// TwinCAT 3 PLC project TcoTixonFeedingTests
// Title: TcoTixonFeedingTests
// Company: Vortex.Library
// Author: TcOpenGroup
// ProjectVersion: 0.6.0.913
// ProgramVersion: 3.1.4024.12
// libraries:
//   Tc2_Standard, * (Beckhoff Automation GmbH)
//   Tc2_System, * (Beckhoff Automation GmbH)
//   Tc3_Module, * (Beckhoff Automation GmbH)
//   TcoAbstractions, 0.6.0.913 (Vortex.Library)
//   TcoCore, 0.6.0.913 (Vortex.Library)
//   TcoIo, 0.6.0.913 (Vortex.Library)
//   TcoTixonFeeding, 0.6.0.913 (Vortex.Library)
//   TcoUtilities, 0.6.0.913 (Vortex.Library)
// project tree:
//   GVLs/ GVL.TcGVL, GVL_iXlinker.TcGVL
//   / PlcTask1.TcTTO
//   POUs/ MAIN.TcPOU
//   Tests/TcoContext/ eTypeOfTixon.TcDUT, SequenceTask.TcPOU, WpfContext.TcPOU
//   Tests/TcoTixonFeeding/ eTcoTixonFeedingSimpleTests.TcDUT, TcoTestContext.TcPOU, TcoTixonFeedingTest.TcPOU
//   DUTs/IO/PDOs/ Channel_830843C1.TcDUT, Channel_42CA91F7.TcDUT
//   DUTs/IO/Boxes/ EK1200_013D0B49.TcDUT, EL1008_78E8D3DD.TcDUT, EL2008_E2806B95.TcDUT, EL9011_D65D3D32.TcDUT
//   DUTs/IO/Devices/ SyncUnitTasks_5FDC9770.TcDUT, SyncUnits_C3A34B50.TcDUT
//   DUTs/IO/Topology/ EK1200_4A80C775.TcDUT, ECAT_x_A7FD7D81.TcDUT
// (motion and I/O tree: see PLC project tcotixonfeeding)
// real-time tasks:
//   TASK PlcTask: cycle T#10ms, priority 20, ADS port 350
//   TASK PlcTask1: cycle T#10ms, priority 1, ADS port 351
//   TASK PN: cycle T#8ms, priority 2, ADS port 301
// variable links:
//   TcoTixonFeedingTests/TcoTixonFeedingTests Instance <-> ECAT
//     PlcTask1 Inputs/GVL_iXlinker.ECAT_x.InfoData.AmsNetId <-> InfoData/AmsNetId
//     PlcTask1 Inputs/GVL_iXlinker.ECAT_x.InfoData.CfgSlaveCount <-> InfoData/CfgSlaveCount
//     PlcTask1 Inputs/GVL_iXlinker.ECAT_x.InfoData.ChangeCount <-> InfoData/ChangeCount
//     PlcTask1 Inputs/GVL_iXlinker.ECAT_x.InfoData.DevId <-> InfoData/DevId
//     PlcTask1 Inputs/GVL_iXlinker.ECAT_x.Inputs.DevState <-> Inputs/DevState
//     PlcTask1 Inputs/GVL_iXlinker.ECAT_x.Inputs.Frm0InputToggle <-> Inputs/Frm0InputToggle
//     PlcTask1 Inputs/GVL_iXlinker.ECAT_x.Inputs.Frm0State <-> Inputs/Frm0State
//     PlcTask1 Inputs/GVL_iXlinker.ECAT_x.Inputs.Frm0WcState <-> Inputs/Frm0WcState
//     PlcTask1 Inputs/GVL_iXlinker.ECAT_x.Inputs.SlaveCount <-> Inputs/SlaveCount
//     PlcTask1 Outputs/GVL_iXlinker.ECAT_x.Outputs.DevCtrl <-> Outputs/DevCtrl
//     PlcTask1 Outputs/GVL_iXlinker.ECAT_x.Outputs.Frm0Ctrl <-> Outputs/Frm0Ctrl
//     PlcTask1 Outputs/GVL_iXlinker.ECAT_x.Outputs.Frm0WcCtrl <-> Outputs/Frm0WcCtrl
//   TcoTixonFeedingTests/TcoTixonFeedingTests Instance <-> ECAT/EK1200/IA1
//     PlcTask1 Inputs/GVL_iXlinker.ECAT_x.EK1200.IA1.Channel_{1..8}.Input <-> Channel {1..8}/Input  (8 links)
//     PlcTask1 Inputs/GVL_iXlinker.ECAT_x.EK1200.IA1.InfoData.State <-> InfoData/State
//     PlcTask1 Inputs/GVL_iXlinker.ECAT_x.EK1200.IA1.WcState.InputToggle <-> WcState/InputToggle
//     PlcTask1 Inputs/GVL_iXlinker.ECAT_x.EK1200.IA1.WcState.WcState <-> WcState/WcState
//   TcoTixonFeedingTests/TcoTixonFeedingTests Instance <-> ECAT/EK1200/QA1
//     PlcTask1 Inputs/GVL_iXlinker.ECAT_x.EK1200.QA1.InfoData.State <-> InfoData/State
//     PlcTask1 Inputs/GVL_iXlinker.ECAT_x.EK1200.QA1.WcState.WcState <-> WcState/WcState
//     PlcTask1 Outputs/GVL_iXlinker.ECAT_x.EK1200.QA1.Channel_{1..8}.Output <-> Channel {1..8}/Output  (8 links)

CONFIGURATION TcoTixonFeedingTests
    RESOURCE PLC ON TwinCAT3
        TASK PlcTask1(INTERVAL := T#10ms, PRIORITY := 1);
        PROGRAM MAIN WITH PlcTask1 : MAIN;
    END_RESOURCE
END_CONFIGURATION

// ---- Tests/TcoContext/eTypeOfTixon.TcDUT
{attribute 'qualified_only'}
{attribute 'strict'}
TYPE eTypeOfTixon :
(
    TixonStep := 0,
    TixonVibro := 1,
    TixonPickStep := 2,
    TixonPickVibro := 3,
    TixonPickVibroBasic := 4
);
END_TYPE

// ---- Tests/TcoTixonFeeding/eTcoTixonFeedingSimpleTests.TcDUT
{attribute 'qualified_only'}
{attribute 'strict'}
TYPE eTcoTixonFeedingSimpleTests :
(
    Restore := 1,
    CleanUp,
    Message,
    PowerDisable,
    PowerEnable,
    Reset,
    Last
);
END_TYPE

// ---- DUTs/IO/PDOs/Channel_830843C1.TcDUT
{attribute 'GeneratedUsingTerminal: EL1008-0000-0018'}
{attribute addProperty BoxType "EL1008-0000-0018"}
{attribute addProperty Id "InputAT %I*BOOL1"}
{attribute addProperty CRC "2198356929"}
{attribute addProperty Size "1"}
TYPE Channel_830843C1 EXTENDS TcoIo.InputBase_8311D824 :
STRUCT
    {attribute addProperty Name "Input"}
    Input AT %I* : BOOL;
END_STRUCT
END_TYPE

// ---- DUTs/IO/PDOs/Channel_42CA91F7.TcDUT
{attribute 'GeneratedUsingTerminal: EL2008-0000-0018'}
{attribute addProperty BoxType "EL2008-0000-0018"}
{attribute addProperty Id "OutputAT %Q*BOOL1"}
{attribute addProperty CRC "1120571895"}
{attribute addProperty Size "1"}
TYPE Channel_42CA91F7 EXTENDS TcoIo.OutputBase_10CEE7DE :
STRUCT
    {attribute addProperty Name "Output"}
    Output AT %Q* : BOOL;
END_STRUCT
END_TYPE

// ---- DUTs/IO/Boxes/EK1200_013D0B49.TcDUT
{attribute 'GeneratedUsingTerminal: EK1200-1388-0000'}
{attribute addProperty VendorId "#x00000002"}
{attribute addProperty BoxType "EK1200-1388-0000"}
{attribute addProperty Description "EK1200-5000 EtherCAT Power supply (2A E-Bus)"}
{attribute addProperty Physics "YK"}
{attribute addProperty Id "EK1200"}
{attribute addProperty CRC "20777801"}
{attribute addProperty Size "0"}
TYPE EK1200_013D0B49 EXTENDS TcoIo.EtcSlaveBoxBase_77A0E4A7 :
STRUCT
END_STRUCT
END_TYPE

// ---- DUTs/IO/Boxes/EL1008_78E8D3DD.TcDUT
{attribute 'GeneratedUsingTerminal: EL1008-0000-0018'}
{attribute addProperty VendorId "#x00000002"}
{attribute addProperty BoxType "EL1008-0000-0018"}
{attribute addProperty Description "EL1008 8Ch. Dig. Input 24V, 3ms"}
{attribute addProperty Physics "KK"}
{attribute addProperty Id "Channel_1AT %I*Channel_830843C11Channel_2AT %I*Channel_830843C11Channel_3AT %I*Channel_830843C11Channel_4AT %I*Channel_830843C11Channel_5AT %I*Channel_830843C11Channel_6AT %I*Channel_830843C11Channel_7AT %I*Channel_830843C11Channel_8AT %I*Channel_830843C11WcStateAT %I*WcState_9091E0EB2InfoDataAT %I*InfoData_6F19DB2B2"}
{attribute addProperty CRC "2028524509"}
{attribute addProperty Size "12"}
TYPE EL1008_78E8D3DD EXTENDS TcoIo.EtcSlaveTerminalBase_947E5A46 :
STRUCT
    {attribute addProperty Name "Channel_1"}
    Channel_1 : Channel_830843C1;
    {attribute addProperty Name "Channel_2"}
    Channel_2 : Channel_830843C1;
    {attribute addProperty Name "Channel_3"}
    Channel_3 : Channel_830843C1;
    {attribute addProperty Name "Channel_4"}
    Channel_4 : Channel_830843C1;
    {attribute addProperty Name "Channel_5"}
    Channel_5 : Channel_830843C1;
    {attribute addProperty Name "Channel_6"}
    Channel_6 : Channel_830843C1;
    {attribute addProperty Name "Channel_7"}
    Channel_7 : Channel_830843C1;
    {attribute addProperty Name "Channel_8"}
    Channel_8 : Channel_830843C1;
    {attribute addProperty Name "WcState"}
    WcState : TcoIo.WcState_9091E0EB;
    {attribute addProperty Name "InfoData"}
    InfoData : TcoIo.InfoData_6F19DB2B;
END_STRUCT
END_TYPE

// ---- DUTs/IO/Boxes/EL2008_E2806B95.TcDUT
{attribute 'GeneratedUsingTerminal: EL2008-0000-0018'}
{attribute addProperty VendorId "#x00000002"}
{attribute addProperty BoxType "EL2008-0000-0018"}
{attribute addProperty Description "EL2008 8Ch. Dig. Output 24V, 0.5A"}
{attribute addProperty Physics "KK"}
{attribute addProperty Id "Channel_1AT %Q*Channel_42CA91F71Channel_2AT %Q*Channel_42CA91F71Channel_3AT %Q*Channel_42CA91F71Channel_4AT %Q*Channel_42CA91F71Channel_5AT %Q*Channel_42CA91F71Channel_6AT %Q*Channel_42CA91F71Channel_7AT %Q*Channel_42CA91F71Channel_8AT %Q*Channel_42CA91F71WcStateAT %I*WcState_0B2B16F91InfoDataAT %I*InfoData_6F19DB2B2"}
{attribute addProperty CRC "3800066965"}
{attribute addProperty Size "11"}
TYPE EL2008_E2806B95 EXTENDS TcoIo.EtcSlaveTerminalBase_947E5A46 :
STRUCT
    {attribute addProperty Name "Channel_1"}
    Channel_1 : Channel_42CA91F7;
    {attribute addProperty Name "Channel_2"}
    Channel_2 : Channel_42CA91F7;
    {attribute addProperty Name "Channel_3"}
    Channel_3 : Channel_42CA91F7;
    {attribute addProperty Name "Channel_4"}
    Channel_4 : Channel_42CA91F7;
    {attribute addProperty Name "Channel_5"}
    Channel_5 : Channel_42CA91F7;
    {attribute addProperty Name "Channel_6"}
    Channel_6 : Channel_42CA91F7;
    {attribute addProperty Name "Channel_7"}
    Channel_7 : Channel_42CA91F7;
    {attribute addProperty Name "Channel_8"}
    Channel_8 : Channel_42CA91F7;
    {attribute addProperty Name "WcState"}
    WcState : TcoIo.WcState_0B2B16F9;
    {attribute addProperty Name "InfoData"}
    InfoData : TcoIo.InfoData_6F19DB2B;
END_STRUCT
END_TYPE

// ---- DUTs/IO/Boxes/EL9011_D65D3D32.TcDUT
{attribute 'GeneratedUsingTerminal: EL9011--0000'}
{attribute addProperty VendorId "#x00000002"}
{attribute addProperty BoxType "EL9011--0000"}
{attribute addProperty Description "EL9011 End Terminal"}
{attribute addProperty Physics ""}
{attribute addProperty Id "EL9011"}
{attribute addProperty CRC "3596434738"}
{attribute addProperty Size "0"}
TYPE EL9011_D65D3D32 EXTENDS TcoIo.EtcSlaveEndTerminalBase_866C7F0C :
STRUCT
END_STRUCT
END_TYPE

// ---- DUTs/IO/Devices/SyncUnitTasks_5FDC9770.TcDUT
{attribute 'GeneratedUsingTerminal: '}
{attribute addProperty BoxType ""}
{attribute addProperty Id "unreferencedAT %I*SyncUnitTask_AB2F50799PlcTask1AT %I*SyncUnitTask_AB2F50799"}
{attribute addProperty CRC "1608292208"}
{attribute addProperty Size "18"}
TYPE SyncUnitTasks_5FDC9770 EXTENDS TcoIo.SyncUnitTasksBase_7C8711EB :
STRUCT
    {attribute addProperty Name "unreferenced"}
    unreferenced : TcoIo.SyncUnitTask_AB2F5079;
    {attribute addProperty Name "PlcTask1"}
    PlcTask1 : TcoIo.SyncUnitTask_AB2F5079;
END_STRUCT
END_TYPE

// ---- DUTs/IO/Devices/SyncUnits_C3A34B50.TcDUT
{attribute 'GeneratedUsingTerminal: '}
{attribute addProperty BoxType ""}
{attribute addProperty Id "_defaultAT %I*SyncUnitTasks_5FDC977018"}
{attribute addProperty CRC "3282258768"}
{attribute addProperty Size "18"}
TYPE SyncUnits_C3A34B50 EXTENDS TcoIo.SyncUnitsBase_AD6C35CE :
STRUCT
    {attribute addProperty Name "_default"}
    _default : SyncUnitTasks_5FDC9770;
END_STRUCT
END_TYPE

// ---- DUTs/IO/Topology/EK1200_4A80C775.TcDUT
{attribute 'GeneratedUsingTerminal: EK1200-1388-0000'}
{attribute addProperty BoxType "EK1200-1388-0000"}
{attribute addProperty Id "IA1EL1008_78E8D3DD12QA1EL2008_E2806B9511Term_4_EL9011EL9011_D65D3D320"}
{attribute addProperty CRC "1249953653"}
{attribute addProperty Size "23"}
{attribute addProperty Name "EK1200"}
TYPE EK1200_4A80C775 EXTENDS EK1200_013D0B49 :
STRUCT
    {attribute addProperty Name "IA1"}
    {attribute addProperty PreviousPort "EK1200 : B"}
    {attribute addProperty SyncUnit "default"}
    IA1 : EL1008_78E8D3DD;
    {attribute addProperty Name "QA1"}
    {attribute addProperty PreviousPort "IA1 : B"}
    {attribute addProperty SyncUnit "default"}
    QA1 : EL2008_E2806B95;
    {attribute addProperty Name "Term 4 (EL9011)"}
    {attribute addProperty PreviousPort "QA1 : B"}
    {attribute addProperty SyncUnit "default"}
    Term_4_EL9011 : EL9011_D65D3D32;
END_STRUCT
END_TYPE

// ---- DUTs/IO/Topology/ECAT_x_A7FD7D81.TcDUT
{attribute 'GeneratedUsingTerminal: IODEVICETYPE_ETHERCATPROT'}
{attribute addProperty BoxType "IODEVICETYPE_ETHERCATPROT"}
{attribute addProperty Id "EK1200EK1200_4A80C77523SyncUnitsSyncUnits_C3A34B5018InputsInputs_A65FACA410OutputsOutputs_23C0ED1D6InfoDataInfoData_84133AC922"}
{attribute addProperty CRC "2818407809"}
{attribute addProperty Size "79"}
{attribute addProperty Name "ECAT"}
TYPE ECAT_x_A7FD7D81 EXTENDS TcoIo.EtcMasterBase_62654B43 :
STRUCT
    {attribute addProperty Name "EK1200"}
    {attribute addProperty PreviousPort "ECAT : Master"}
    {attribute addProperty SyncUnit "default"}
    EK1200 : EK1200_4A80C775;
    {attribute addProperty Name "SyncUnits"}
    SyncUnits : SyncUnits_C3A34B50;
    {attribute addProperty Name "Inputs"}
    Inputs : TcoIo.Inputs_A65FACA4;
    {attribute addProperty Name "Outputs"}
    Outputs : TcoIo.Outputs_23C0ED1D;
    {attribute addProperty Name "InfoData"}
    InfoData : TcoIo.InfoData_84133AC9;
END_STRUCT
END_TYPE

// ---- GVLs/GVL.TcGVL
{attribute 'qualified_only'}
VAR_GLOBAL
END_VAR

// ---- GVLs/GVL_iXlinker.TcGVL
{attribute 'qualified_only'}
VAR_GLOBAL
    ECAT_x : ECAT_x_A7FD7D81;
END_VAR

// ---- POUs/MAIN.TcPOU
PROGRAM MAIN
VAR
    _tcoTestContext : TcoTestContext;
    _wpfContext : WpfContext;
    _wpfContextCall : BOOL := FALSE;
END_VAR

_tcoTestContext.ProbeRun();

IF _wpfContextCall THEN
    _wpfContext.Run();
END_IF

END_PROGRAM

// ---- Tests/TcoTixonFeeding/TcoTestContext.TcPOU
FUNCTION_BLOCK TcoTestContext EXTENDS TcoCore._internals_TcoContext
VAR
    _sut : TcoTixonFeedingTest(THIS^);
    _callMyPlcInstance : BOOL := FALSE;
    _enable : BOOL;
    _enablePositive : BOOL;
    _enableNegative : BOOL;
    _calibrationCam : BOOL;
    _position : LREAL;
    _velocity : LREAL;
    _acceleration : LREAL;
    _deceleration : LREAL;
    _jerk : LREAL;
    _inString : STRING;
    _done : BOOL;
    _arranged : BOOL;
    _axisReferenceType : INT;
END_VAR

METHOD PROTECTED Main
//_sut(inEnable := _enable,
//    inEnablePositive := _enablePositive,
//    inEnableNegative := _enableNegative,
//    inCalibrationCam := _calibrationCam,
//    inoAxisRef := GVL.Axis1);
//
//CASE _testId OF
//    eTcoDriveSimpleTests.Restore:
//        _sut.Restore();
//    eTcoDriveSimpleTests.CleanUp:
//        _sut._messenger.Clear();
//    {region "T003_Message"}
//    eTcoDriveSimpleTests.Message:
//        _sut.Messenger.Error(_inString);
//        _done := _plcCycleCounter > 1;
//        ProbeDoneWhen(_done);
//    {endregion}
//    {region "T004_PowerDisable"}
//    eTcoDriveSimpleTests.PowerDisable:
//        _enable := FALSE;
//        _done := _sut._axisStatus.Disabled; // OR _plcCycleCounter > 1;
//        ProbeDoneWhen(_done);
//    {endregion}
//    {region "T005_PowerEnable"}
//    eTcoDriveSimpleTests.PowerEnable:
//        _enable := TRUE;
//        _done := _sut._axisStatus.Operational; // OR _plcCycleCounter > 15;
//        ProbeDoneWhen(_done);
//    {endregion}
//    {region "T006_Reset"}
//    eTcoDriveSimpleTests.Reset:
//        IF NOT _arranged THEN
//            _sut.MoveRelative(inDistance := 500,
//                inVelocity := 50000000,
//                inAcceleration := -1,
//                inDeceleration := -1,
//                inJerk := -1);
//
//            IF _sut._axisStatus.Error THEN
//                _arranged := true;
//            END_IF
//
//            RETURN;
//        END_IF
//
//        _sut.Reset();
//        _done := _sut.ResetTask.Done OR _sut.ResetTask.Error; // OR _plcCycleCounter > 1;
//        ProbeDoneWhen(_done);
//    {endregion}
//    {region "T007_MoveRelativePositiveWithDisabledPositiveDirection"}
//    eTcoDriveSimpleTests.MoveRelativePositiveWithDisabledPositiveDirection:
//        IF NOT _arranged THEN
//            _enable := TRUE;
//            _enablePositive := FALSE;
//            _enableNegative := FALSE;
//
//            IF _sut._axisStatus.Operational THEN
//                _arranged := TRUE;
//            END_IF
//
//            RETURN;
//        END_IF;
//
//        _sut.MoveRelative(inDistance := _position,
//            inVelocity := _velocity,
//            inAcceleration := _acceleration,
//            inDeceleration := _deceleration,
//            inJerk := _jerk);
//
//        _done := _sut.MoveRelativeTask.Done OR _sut.MoveRelativeTask.Error; // OR _sut._axisStatus.Error;// OR _plcCycleCounter > 5;
//        ProbeDoneWhen(_done);
//    {endregion}
//    {region "T008_MoveRelativePositiveWithEnabledPositiveDirection"}
//    eTcoDriveSimpleTests.MoveRelativePositiveWithEnabledPositiveDirection:
//        IF NOT _arranged THEN
//            _enable := TRUE;
//            _enablePositive := TRUE;
//            _enableNegative := FALSE;
//
//            IF _sut._axisStatus.Operational THEN
//                _arranged := TRUE;
//            END_IF
//
//            RETURN;
//        END_IF;
//
//        _sut.MoveRelative(inDistance := _position,
//            inVelocity := _velocity,
//            inAcceleration := _acceleration,
//            inDeceleration := _deceleration,
//            inJerk := _jerk);
//
//        _done := _sut.MoveRelativeTask.Done OR _sut.MoveRelativeTask.Error; // OR  _plcCycleCounter > 1000;
//        ProbeDoneWhen(_done);
//    {endregion}
//    {region "T009_MoveRelativeNegativeWithDisabledNegativeDirection"}
//    eTcoDriveSimpleTests.MoveRelativeNegativeWithDisabledNegativeDirection:
//        IF NOT _arranged THEN
//            _enable := TRUE;
//            _enablePositive := FALSE;
//            _enableNegative := FALSE;
//
//            IF _sut._axisStatus.Operational THEN
//                _arranged := TRUE;
//            END_IF
//
//            RETURN;
//        END_IF;
//
//        _sut.MoveRelative(inDistance := _position,
//            inVelocity := _velocity,
//            inAcceleration := _acceleration,
//            inDeceleration := _deceleration,
//            inJerk := _jerk);
//
//        _done := _sut.MoveRelativeTask.Done OR _sut.MoveRelativeTask.Error; // OR _sut._axisStatus.Error;// OR _plcCycleCounter > 5;
//        ProbeDoneWhen(_done);
//    {endregion}
//    {region "T010_MoveRelativeNegativeWithEnabledNegativeDirection"}
//    eTcoDriveSimpleTests.MoveRelativeNegativeWithEnabledNegativeDirection:
//        IF NOT _arranged THEN
//            _enable := TRUE;
//            _enablePositive := TRUE;
//            _enableNegative := TRUE;
//
//            IF _sut._axisStatus.Operational THEN
//                _arranged := TRUE;
//            END_IF
//
//            RETURN;
//        END_IF;
//
//        _sut.MoveRelative(inDistance := _position,
//            inVelocity := _velocity,
//            inAcceleration := _acceleration,
//            inDeceleration := _deceleration,
//            inJerk := _jerk);
//
//        _done := _sut.MoveRelativeTask.Done OR _sut.MoveRelativeTask.Error; // OR  _plcCycleCounter > 1000;
//        ProbeDoneWhen(_done);
//    {endregion}
//    {region "T011_HommingDirect"}
//    eTcoDriveSimpleTests.HommingDirect:
//        IF NOT _arranged THEN
//            _enable := TRUE;
//            _enablePositive := FALSE;
//            _enableNegative := TRUE;
//
//            IF _sut._axisStatus.Operational THEN
//                _arranged := TRUE;
//            END_IF
//
//            RETURN;
//        END_IF;
//
//        _sut.Home(inPosition := _position,
//            inHomingMode := TcoDrivesBeckhoff.eHomingMode.MC_Direct,
//            inClearPositionLag := FALSE,
//            inSearchDirection := TcoDrivesBeckhoff.eDirection.MC_Undefined_Direction,
//            inSearchVelocity := _velocity,
//            inSyncDirection := TcoDrivesBeckhoff.eDirection.MC_Undefined_Direction,
//            inSyncVelocity := _velocity,
//            inReferenceMode := TcoDrivesBeckhoff.eEncoderReferenceMode.ENCODERREFERENCEMODE_DEFAULT);
//
//        _done := _sut.HomeTask.Done OR _sut.HomeTask.Error; //OR _plcCycleCounter > 1000;
//        ProbeDoneWhen(_done);
//    {endregion}
//    {region "T012_MoveVelocityPositiveWithDisabledPositiveDirection"}
//    eTcoDriveSimpleTests.MoveVelocityPositiveWithDisabledPositiveDirection:
//        IF NOT _arranged THEN
//            _enable := TRUE;
//            _enablePositive := FALSE;
//            _enableNegative := FALSE;
//
//            IF _sut._axisStatus.Operational THEN
//                _arranged := TRUE;
//            END_IF
//
//            RETURN;
//        END_IF;
//
//        _sut.MoveVelocity(inVelocity := _velocity,
//            inAcceleration := _acceleration,
//            inDeceleration := _deceleration,
//            inJerk := _jerk,
//            inDirection := TcoDrivesBeckhoff.eDirection.MC_Positive_Direction);
//
//        _done := _sut.MoveVelocityTask.Done OR _sut.MoveVelocityTask.Error; // OR  _sut._axisStatus.Error;// OR _plcCycleCounter > 5;
//        ProbeDoneWhen(_done);
//    {endregion}
//    {region "T013_MoveVelocityPositiveWithEnabledPositiveDirection"}
//    eTcoDriveSimpleTests.MoveVelocityPositiveWithEnabledPositiveDirection:
//        IF NOT _arranged THEN
//            _enable := TRUE;
//            _enablePositive := TRUE;
//            _enableNegative := FALSE;
//
//            IF _sut._axisStatus.Operational THEN
//                _arranged := TRUE;
//            END_IF
//
//            RETURN;
//        END_IF;
//
//        _sut.MoveVelocity(inVelocity := _velocity,
//            inAcceleration := _acceleration,
//            inDeceleration := _deceleration,
//            inJerk := _jerk,
//            inDirection := TcoDrivesBeckhoff.eDirection.MC_Positive_Direction);
//
//        _done := _sut.MoveVelocityTask.Done OR _sut.MoveVelocityTask.Error; // OR  _plcCycleCounter > 1000;
//        ProbeDoneWhen(_done);
//    {endregion}
//    {region "T014_Stop"}
//    eTcoDriveSimpleTests.Stop:
//        IF NOT _arranged THEN
//            _enable := TRUE;
//            _enablePositive := TRUE;
//            _enableNegative := TRUE;
//
//            IF _sut._axisStatus.Operational THEN
//                _arranged := TRUE;
//            END_IF
//
//            RETURN;
//        END_IF;
//
//        _sut.Stop(inDeceleration := _deceleration, inJerk := _jerk);
//        _done := _sut.StopTask.Done OR _sut.StopTask.Error; // OR  _plcCycleCounter > 1000;
//        ProbeDoneWhen(_done);
//    {endregion}
//    {region "T015_MoveVelocityNegativeWithDisabledNegativeDirection"}
//    eTcoDriveSimpleTests.MoveVelocityNegativeWithDisabledNegativeDirection:
//        IF NOT _arranged THEN
//            _enable := TRUE;
//            _enablePositive := FALSE;
//            _enableNegative := FALSE;
//
//            IF _sut._axisStatus.Operational THEN
//                _arranged := TRUE;
//            END_IF
//
//            RETURN;
//        END_IF;
//
//        _sut.MoveVelocity(inVelocity := _velocity,
//            inAcceleration := _acceleration,
//            inDeceleration := _deceleration,
//            inJerk := _jerk,
//            inDirection := TcoDrivesBeckhoff.eDirection.MC_Negative_Direction);
//
//        _done := _sut.MoveVelocityTask.Done OR _sut.MoveVelocityTask.Error; // OR  _sut._axisStatus.Error;// OR _plcCycleCounter > 5;
//        ProbeDoneWhen(_done);
//    {endregion}
//    {region "T016_MoveVelocityNegativeWithEnabledNegativeDirection"}
//    eTcoDriveSimpleTests.MoveVelocityNegativeWithEnabledNegativeDirection:
//        IF NOT _arranged THEN
//            _enable := TRUE;
//            _enablePositive := FALSE;
//            _enableNegative := TRUE;
//
//            IF _sut._axisStatus.Operational THEN
//                _arranged := TRUE;
//            END_IF
//
//            RETURN;
//        END_IF;
//
//        _sut.MoveVelocity(inVelocity := _velocity,
//            inAcceleration := _acceleration,
//            inDeceleration := _deceleration,
//            inJerk := _jerk,
//            inDirection := TcoDrivesBeckhoff.eDirection.MC_Negative_Direction);
//
//        _done := _sut.MoveVelocityTask.Done OR _sut.MoveVelocityTask.Error; // OR  _plcCycleCounter > 1000;
//        ProbeDoneWhen(_done);
//    {endregion}
//    {region "T017_MoveAbsoluteDisabled"}
//    eTcoDriveSimpleTests.MoveAbsoluteDisabled:
//        IF NOT _arranged THEN
//            _enable := FALSE;
//            _enablePositive := FALSE;
//            _enableNegative := FALSE;
//            _arranged := TRUE;
//            RETURN;
//        END_IF;
//
//        _sut.MoveAbsolute(inPosition := _position,
//            inVelocity := _velocity,
//            inAcceleration := _acceleration,
//            inDeceleration := _deceleration,
//            inJerk := _jerk);
//
//        _done := _sut.MoveAbsoluteTask.Done OR _sut.MoveAbsoluteTask.Error OR _plcCycleCounter > 10;
//        ProbeDoneWhen(_done);
//	{endregion}
//    {region "T018_MoveAbsoluteDisabledPositiveDirection"}
//    eTcoDriveSimpleTests.MoveAbsoluteDisabledPositiveDirection:
//        IF NOT _arranged THEN
//            _enable := TRUE;
//            _enablePositive := FALSE;
//            _enableNegative := TRUE;
//            _arranged := TRUE;
//            RETURN;
//        END_IF;
//
//        _sut.MoveAbsolute(inPosition := _position,
//            inVelocity := _velocity,
//            inAcceleration := _acceleration,
//            inDeceleration := _deceleration,
//            inJerk := _jerk);
//
//        _done := _sut.MoveAbsoluteTask.Done OR _sut.MoveAbsoluteTask.Error; // OR _sut._axisStatus.Error;// OR _plcCycleCounter > 5;
//        ProbeDoneWhen(_done);
//	{endregion}
//    {region "T019_MoveAbsoluteEnabledPositiveDirection"}
//    eTcoDriveSimpleTests.MoveAbsoluteEnabledPositiveDirection:
//        IF NOT _arranged THEN
//            _enable := TRUE;
//            _enablePositive := TRUE;
//            _enableNegative := FALSE;
//            _arranged := TRUE;
//            RETURN;
//        END_IF;
//
//        _sut.MoveAbsolute(inPosition := _position,
//            inVelocity := _velocity,
//            inAcceleration := _acceleration,
//            inDeceleration := _deceleration,
//            inJerk := _jerk);
//
//        _done := _sut.MoveAbsoluteTask.Done OR _sut.MoveAbsoluteTask.Error; // OR _sut._axisStatus.Error;// OR _plcCycleCounter > 5;
//        ProbeDoneWhen(_done);
//	{endregion}
//    {region "T020_MoveAbsoluteDisabledNegativeDirection"}
//    eTcoDriveSimpleTests.MoveAbsoluteDisabledNegativeDirection:
//        IF NOT _arranged THEN
//            _enable := TRUE;
//            _enablePositive := FALSE;
//            _enableNegative := FALSE;
//            _arranged := TRUE;
//            RETURN;
//        END_IF;
//
//        _sut.MoveAbsolute(inPosition := _position,
//            inVelocity := _velocity,
//            inAcceleration := _acceleration,
//            inDeceleration := _deceleration,
//            inJerk := _jerk);
//
//        _done := _sut.MoveAbsoluteTask.Done OR _sut.MoveAbsoluteTask.Error; // OR _sut._axisStatus.Error;// OR _plcCycleCounter > 5;
//        ProbeDoneWhen(_done);
//	{endregion}
//    {region "T021_MoveAbsoluteEnabledNegativeDirection"}
//    eTcoDriveSimpleTests.MoveAbsoluteEnabledNegativeDirection:
//        IF NOT _arranged THEN
//            _enable := TRUE;
//            _enablePositive := FALSE;
//            _enableNegative := TRUE;
//            _arranged := TRUE;
//            RETURN;
//        END_IF;
//
//        _sut.MoveAbsolute(inPosition := _position,
//            inVelocity := _velocity,
//            inAcceleration := _acceleration,
//            inDeceleration := _deceleration,
//            inJerk := _jerk);
//
//        _done := _sut.MoveAbsoluteTask.Done OR _sut.MoveAbsoluteTask.Error; // OR _sut._axisStatus.Error;// OR _plcCycleCounter > 5;
//        ProbeDoneWhen(_done);
//	{endregion}
//END_CASE
END_METHOD

END_FUNCTION_BLOCK

// ---- Tests/TcoTixonFeeding/TcoTixonFeedingTest.TcPOU
FUNCTION_BLOCK TcoTixonFeedingTest EXTENDS TcoTixonFeeding.TcoTixonStep_v_1_x_x
VAR
    _serviceModeCount : ULINT;
    _serviceModeOverride : LREAL;
END_VAR
VAR
END_VAR

//SUPER^(	inEnable 			:=	inEnable,
//		inEnablePositive	:=	inEnablePositive,
//		inEnableNegative	:=	inEnableNegative,
//		inCalibrationCam	:=	inCalibrationCam,
//		inoAxisRef			:=	inoAxisRef);
//

END_FUNCTION_BLOCK

// ---- Tests/TcoContext/WpfContext.TcPOU
FUNCTION_BLOCK WpfContext EXTENDS TcoCore.TcoContext
VAR
    _serviceModeActive : BOOL;
    {attribute addProperty Name "<#TcoTixonStep #>"}
    _tixonStepFeeder : TcoTixonFeeding.TcoTixonStep_v_1_x_x(THIS^);
    {attribute addProperty Name "<#TcoTixonVibro #>"}
    _tixonVibroFeeder : TcoTixonFeeding.TcoTixonVibro_v_1_x_x(THIS^);
    {attribute addProperty Name "<#TcoTixonPickVibro #>"}
    _tixonPickVibroFeeder : TcoTixonFeeding.TcoTixonPickVibro_v_1_x_x(THIS^);
    {attribute addProperty Name "<#TcoTixonPickStep #>"}
    _tixonPickStepFeeder : TcoTixonFeeding.TcoTixonPickStep_v_1_x_x(THIS^);
    {attribute addProperty Name "<#TcoTixonPickVibroBasic #>"}
    _tixonPickVibroBasicFeeder : TcoTixonFeeding.TcoTixonPickVibroBasic_v_1_x_x(THIS^);
    _dialogTixon : TcoCore.TcoDialog(THIS^);
    _sequenceTixonStep : TcoCore.TcoSequence(THIS^, eRestoreMode.None);
    _observerTixonStep : TcoCore.TcoSequencerObserver(THIS^);
    {attribute addProperty Name "Start sequence Step"}
    _sequenceTixonStepTask : SequenceTask(THIS^);
    {attribute addProperty Name "Requred attempts Step"}
    _maxAllowedAttemptsTixonStep : INT;
    _sequenceTixonVibro : TcoCore.TcoSequence(THIS^, eRestoreMode.None);
    _observerTixonVibro : TcoCore.TcoSequencerObserver(THIS^);
    {attribute addProperty Name "Start sequence Vibro"}
    _sequenceTixonVibroTask : SequenceTask(THIS^);
    {attribute addProperty Name "Requred attempts Vibro"}
    _maxAllowedAttemptsTixonVibro : INT;
    _sequenceTixonPickVibro : TcoCore.TcoSequence(THIS^, eRestoreMode.None);
    _observerTixonPickVibro : TcoCore.TcoSequencerObserver(THIS^);
    {attribute addProperty Name "Start sequence PickVibro"}
    _sequenceTixonPickVibroTask : SequenceTask(THIS^);
    {attribute addProperty Name "Requred attempts PickVibro"}
    _maxAllowedAttemptsTixonPickVibro : INT;
    _sequenceTixonPickStep : TcoCore.TcoSequence(THIS^, eRestoreMode.None);
    _observerTixonPickStep : TcoCore.TcoSequencerObserver(THIS^);
    {attribute addProperty Name "Start sequence PickStep"}
    _sequenceTixonPickStepTask : SequenceTask(THIS^);
    {attribute addProperty Name "Requred attempts PickStep"}
    _maxAllowedAttemptsTixonPickStep : INT;
    _sequenceTixonPickVibroBasic : TcoCore.TcoSequence(THIS^, eRestoreMode.None);
    _observerTixonPickVibroBasic : TcoCore.TcoSequencerObserver(THIS^);
    {attribute addProperty Name "Start sequence Vibro"}
    _sequenceTixonPickVibroBasicTask : SequenceTask(THIS^);
    {attribute addProperty Name "Requred attempts Vibro"}
    _maxAllowedAttemptsTixonPickVibroBasic : INT;
    {attribute addProperty Name "TYPE OF TIXON "}
    _testedTixon : eTypeOfTixon;
    {attribute addProperty Name "ESTIMATED CYCLE TIME"}
    _estimatedCycleTime : TIME;
    {attribute addProperty Name "PUSH(SHOT) CYCLE TIME"}
    _pushTime : TIME;
    {attribute addProperty Name "ACTUAL COUNT"}
    _actualAttempt : DINT;
END_VAR

(*~
    <docu>
        <summary>
            Main method of the TcoContext. This is the entry point of any control logic that belongs to this context.
            The call of this method is ensured by calling the <c>InstanceName.Run()</c> method, and it must not be called explicitly.
            This method is abstract, and it must be overridden in derived block.
        </summary>
    </docu>
~*)
METHOD PROTECTED Main
IF _serviceModeActive THEN
    _tixonStepFeeder.Service();
END_IF

CASE _testedTixon OF
    eTypeOfTixon.TixonStep:
        _tixonStepFeeder(inControllerInAuto := GVL_iXlinker.ECAT_x.EK1200.IA1.Channel_1.Input,
            inNotEmptyFeeder := GVL_iXlinker.ECAT_x.EK1200.IA1.Channel_2.Input,
            inSeparatorHomePos := GVL_iXlinker.ECAT_x.EK1200.IA1.Channel_3.Input,
            inFillingSensor := GVL_iXlinker.ECAT_x.EK1200.IA1.Channel_4.Input,
            inSeparatorPresent := GVL_iXlinker.ECAT_x.EK1200.IA1.Channel_5.Input,
            inStepperHomePos := GVL_iXlinker.ECAT_x.EK1200.IA1.Channel_6.Input,
            inStepperWorkPos := GVL_iXlinker.ECAT_x.EK1200.IA1.Channel_7.Input,
            inComponentOutOfBox := GVL_iXlinker.ECAT_x.EK1200.IA1.Channel_8.Input,
            //inSeparatorWorkPos:=GVL_iXlinker.ECAT_x.EK1200.IA1.Channel_9.Input ,
            outFeedingA => GVL_iXlinker.ECAT_x.EK1200.qA1.Channel_1.Output,
            outSepareComponent => GVL_iXlinker.ECAT_x.EK1200.qA1.Channel_2.Output,
            outBlowValveA => GVL_iXlinker.ECAT_x.EK1200.qA1.Channel_3.Output,
            outRedLed => GVL_iXlinker.ECAT_x.EK1200.qA1.Channel_4.Output,
            outGreenLed => GVL_iXlinker.ECAT_x.EK1200.qA1.Channel_5.Output,
            outHopper => GVL_iXlinker.ECAT_x.EK1200.qA1.Channel_6.Output,
            outStepperValve => GVL_iXlinker.ECAT_x.EK1200.qA1.Channel_7.Output,
            outShotComponent => GVL_iXlinker.ECAT_x.EK1200.qA1.Channel_8.Output);

        _tixonStepFeeder.Service();
    eTypeOfTixon.TixonVibro:
        _tixonVibroFeeder(inControllerInAuto := GVL_iXlinker.ECAT_x.EK1200.IA1.Channel_1.Input,
            inNotEmptyFeeder := GVL_iXlinker.ECAT_x.EK1200.IA1.Channel_2.Input,
            inSeparatorHomePos := GVL_iXlinker.ECAT_x.EK1200.IA1.Channel_3.Input,
            inFillingSensor := GVL_iXlinker.ECAT_x.EK1200.IA1.Channel_4.Input,
            inSeparatorPresent := GVL_iXlinker.ECAT_x.EK1200.IA1.Channel_5.Input,
            inComponentOutOfBox := GVL_iXlinker.ECAT_x.EK1200.IA1.Channel_6.Input,
            inSeparatorWorkPos := GVL_iXlinker.ECAT_x.EK1200.IA1.Channel_7.Input,
            outFeedingA => GVL_iXlinker.ECAT_x.EK1200.qA1.Channel_1.Output,
            outSepareComponent => GVL_iXlinker.ECAT_x.EK1200.qA1.Channel_2.Output,
            outBlowValveA => GVL_iXlinker.ECAT_x.EK1200.qA1.Channel_3.Output,
            outRedLed => GVL_iXlinker.ECAT_x.EK1200.qA1.Channel_4.Output,
            outGreenLed => GVL_iXlinker.ECAT_x.EK1200.qA1.Channel_5.Output,
            outHopper => GVL_iXlinker.ECAT_x.EK1200.qA1.Channel_6.Output,
            outShotComponent => GVL_iXlinker.ECAT_x.EK1200.qA1.Channel_7.Output);

        _tixonVibroFeeder.Service();
    eTypeOfTixon.TixonPickStep:
        _tixonPickStepFeeder(inControllerInAuto := GVL_iXlinker.ECAT_x.EK1200.IA1.Channel_1.Input,
            inNotEmptyFeeder := GVL_iXlinker.ECAT_x.EK1200.IA1.Channel_2.Input,
            inSeparatorHomePos := GVL_iXlinker.ECAT_x.EK1200.IA1.Channel_3.Input,
            inFillingSensor := GVL_iXlinker.ECAT_x.EK1200.IA1.Channel_4.Input,
            inSeparatorPresent := GVL_iXlinker.ECAT_x.EK1200.IA1.Channel_5.Input,
            inStepperHomePos := GVL_iXlinker.ECAT_x.EK1200.IA1.Channel_6.Input,
            inStepperWorkPos := GVL_iXlinker.ECAT_x.EK1200.IA1.Channel_7.Input,
            outFeedingA => GVL_iXlinker.ECAT_x.EK1200.qA1.Channel_1.Output,
            outSepareComponent => GVL_iXlinker.ECAT_x.EK1200.qA1.Channel_2.Output,
            outBlowValveA => GVL_iXlinker.ECAT_x.EK1200.qA1.Channel_3.Output,
            outRedLed => GVL_iXlinker.ECAT_x.EK1200.qA1.Channel_4.Output,
            outGreenLed => GVL_iXlinker.ECAT_x.EK1200.qA1.Channel_5.Output,
            outHopper => GVL_iXlinker.ECAT_x.EK1200.qA1.Channel_6.Output,
            outStepperValve => GVL_iXlinker.ECAT_x.EK1200.qA1.Channel_7.Output);

        _tixonPickStepFeeder.Service();
    eTypeOfTixon.TixonPickVibro:
        _tixonPickVibroFeeder(inControllerInAuto := GVL_iXlinker.ECAT_x.EK1200.IA1.Channel_1.Input,
            inNotEmptyFeeder := GVL_iXlinker.ECAT_x.EK1200.IA1.Channel_2.Input,
            inSeparatorHomePos := GVL_iXlinker.ECAT_x.EK1200.IA1.Channel_3.Input,
            inFillingSensor := GVL_iXlinker.ECAT_x.EK1200.IA1.Channel_4.Input,
            inSeparatorPresent := GVL_iXlinker.ECAT_x.EK1200.IA1.Channel_5.Input,
            inSeparatorWorkPos := GVL_iXlinker.ECAT_x.EK1200.IA1.Channel_6.Input,
            outFeedingA => GVL_iXlinker.ECAT_x.EK1200.qA1.Channel_1.Output,
            outSepareComponent => GVL_iXlinker.ECAT_x.EK1200.qA1.Channel_2.Output,
            outBlowValveA => GVL_iXlinker.ECAT_x.EK1200.qA1.Channel_3.Output,
            outRedLed => GVL_iXlinker.ECAT_x.EK1200.qA1.Channel_4.Output,
            outGreenLed => GVL_iXlinker.ECAT_x.EK1200.qA1.Channel_5.Output,
            outHopper => GVL_iXlinker.ECAT_x.EK1200.qA1.Channel_6.Output,
            outFeedingB => GVL_iXlinker.ECAT_x.EK1200.qA1.Channel_7.Output,
            outBlowValveB => GVL_iXlinker.ECAT_x.EK1200.qA1.Channel_8.Output);

        _tixonPickVibroFeeder.Service();
    eTypeOfTixon.TixonPickVibroBasic:
        _tixonPickVibroBasicFeeder(inControllerInAuto := GVL_iXlinker.ECAT_x.EK1200.IA1.Channel_1.Input,
            inNotEmptyFeeder := GVL_iXlinker.ECAT_x.EK1200.IA1.Channel_2.Input,
            inSeparatorHomePos := GVL_iXlinker.ECAT_x.EK1200.IA1.Channel_3.Input,
            inSeparatorPresent := GVL_iXlinker.ECAT_x.EK1200.IA1.Channel_5.Input,
            inSeparatorWorkPos := GVL_iXlinker.ECAT_x.EK1200.IA1.Channel_6.Input,
            outFeedingA => GVL_iXlinker.ECAT_x.EK1200.qA1.Channel_1.Output,
            outSepareComponent => GVL_iXlinker.ECAT_x.EK1200.qA1.Channel_2.Output,
            outBlowValveA => GVL_iXlinker.ECAT_x.EK1200.qA1.Channel_3.Output,
            outRedLed => GVL_iXlinker.ECAT_x.EK1200.qA1.Channel_4.Output,
            outGreenLed => GVL_iXlinker.ECAT_x.EK1200.qA1.Channel_5.Output,
            outHopper => GVL_iXlinker.ECAT_x.EK1200.qA1.Channel_6.Output,);

        _tixonPickVibroBasicFeeder.Service();
END_CASE

_sequenceTixonStepTask.Enabled := _testedTixon = eTypeOfTixon.TixonStep;
_sequenceTixonStepTask(Sequence := _sequenceTixonStep);

IF (_sequenceTixonStepTask.Execute()) THEN
    SequenceTixonStep();
END_IF;

_sequenceTixonVibroTask.Enabled := _testedTixon = eTypeOfTixon.TixonVibro;
_sequenceTixonVIbroTask(Sequence := _sequenceTixonVibro);

IF (_sequenceTixonVibroTask.Execute()) THEN
    SequenceTixonVibro();
END_IF;

_sequenceTixonPickVibroTask.Enabled := _testedTixon = eTypeOfTixon.TixonPickVibro;
_sequenceTixonPickVibroTask(Sequence := _sequenceTixonPickVibro);

IF (_sequenceTixonPickVibroTask.Execute()) THEN
    SequenceTixonPickVibro();
END_IF;

_sequenceTixonPickStepTask.Enabled := _testedTixon = eTypeOfTixon.TixonPickStep;
_sequenceTixonPickStepTask(Sequence := _sequenceTixonPickStep);

IF (_sequenceTixonPickStepTask.Execute()) THEN
    SequenceTixonPickStep();
END_IF;

_sequenceTixonPickVibroBasicTask.Enabled := _testedTixon = eTypeOfTixon.TixonPickVibroBasic;
_sequenceTixonPickVibroBasicTask(Sequence := _sequenceTixonPickVibroBasic);

IF (_sequenceTixonPickVibroBasicTask.Execute()) THEN
    SequenceTixonPickVibroBasic();
END_IF;
END_METHOD

METHOD SequenceTixonPickStep
VAR
    seq : REFERENCE TO TcoCore.TcoSequence;
    answer : TcoCore.eDialogAnswer;
    done : BOOL;
    ProbeDoneWhen : INT;
END_VAR
VAR_INST
    _noOfAttmets : INT;
    _timer : ton;
END_VAR
seq REF= _sequenceTixonStep;
seq.Open();
seq.Observer := _observerTixonStep;
_tixonPickStepFeeder.CyclicBufferFeed();
_tixonPickStepFeeder.CyclicStepperFeed();
_tixonPickStepFeeder.CyclicHopperFeed();
_tixonPickStepFeeder.DefaultSignalisation();
_actualAttempt := _noOfAttmets;

IF (seq.Step(inStepID := 0, inEnabled := TRUE, inStepDescription := 'READY TO START')) THEN
    //--------------------------------------------------------
    _noOfAttmets := 0;

    answer := _dialogTixon.Show()
        .WithType(eDialogType.Question)
        .WithCaption('Ready to go?')
        .WithText('Do you really want to start feeding? Do we go ahead?')
        .WithYesNo().Answer;

    //
    IF (answer = TcoCore.eDialogAnswer.Yes) THEN
        seq.CompleteStep();
    ELSIF (answer = TcoCore.eDialogAnswer.No) THEN
        _sequenceTixonPickStepTask.Restore();
    END_IF;
    //--------------------------------------------------------
END_IF;

IF (seq.Step(inStepID := 10, inEnabled := TRUE, inStepDescription := 'RESTORE')) THEN
    //--------------------------------------------------------
    _tixonPickStepFeeder.Restore();
    seq.CompleteStep();
    //--------------------------------------------------------
END_IF;

IF (seq.Step(inStepID := 11, inEnabled := TRUE, inStepDescription := 'START FEEDING TASK')) THEN
    //--------------------------------------------------------
    seq.StepCompleteWhen(_tixonPickStepFeeder.Separe().Done);
    //--------------------------------------------------------
END_IF;

IF (seq.Step(inStepID := 12, inEnabled := TRUE, inStepDescription := 'WAIT FOR COMPONENT')) THEN
    //--------------------------------------------------------
    IF _tixonPickStepFeeder.Status.ComponentReady THEN
        seq.CompleteStep();
        _timer(IN := FALSE);
    END_IF;
    //--------------------------------------------------------
END_IF;

IF (seq.Step(inStepID := 13, inEnabled := TRUE, inStepDescription := 'WAIT FOR PICK - INTERUPT PICK ZONE')) THEN
    //--------------------------------------------------------
    IF _tixonPickStepFeeder.Status.InPickZone THEN
        seq.CompleteStep();
    END_IF

    //--------------------------------------------------------
END_IF;

IF (seq.Step(inStepID := 14, inEnabled := TRUE, inStepDescription := 'WAIT FOR PICK - RELEASE PICK')) THEN
    //--------------------------------------------------------
    IF NOT _tixonPickStepFeeder.Status.InPickZone AND NOT _tixonPickStepFeeder.Status.SeparatorPresent THEN
        seq.CompleteStep();
    END_IF

    //--------------------------------------------------------
END_IF;

IF (seq.Step(inStepID := 16, inEnabled := TRUE, inStepDescription := 'COUNT')) THEN
    //--------------------------------------------------------
    IF _noOfAttmets < _maxAllowedAttemptsTixonPickStep THEN
        _noOfAttmets := _noOfAttmets + 1;
        seq.RequestStep(11);
    ELSE
        seq.CompleteStep();
    end_if;
    //--------------------------------------------------------
END_IF;

IF (seq.Step(inStepID := 600, inEnabled := TRUE, inStepDescription := 'ASKING FOR RESTORING')) THEN
    //    --------------------------------------------------------
    _tixonPickVibroFeeder.Restore();
    answer := _dialogTixon.Show().WithType(eDialogType.Question).WithCaption('Question?').WithText('Do you want to repat it?').WithYesNo().Answer;

    IF (answer = TcoCore.eDialogAnswer.Yes) THEN
        seq.CompleteStep();
    ELSIF (answer = TcoCore.eDialogAnswer.No) THEN
        _sequenceTixonPickStep.Restore();
    END_IF;
    //    --------------------------------------------------------
END_IF;

IF (seq.Step(inStepID := seq.RESTORE_STEP_ID, inEnabled := TRUE, inStepDescription := 'RETURN TO THE START OF THE SEQUENCE')) THEN
    //--------------------------------------------------------
    seq.CompleteSequence();
    //--------------------------------------------------------
END_IF;

seq.Close();
END_METHOD

METHOD SequenceTixonPickVibro
VAR
    seq : REFERENCE TO TcoCore.TcoSequence;
    answer : TcoCore.eDialogAnswer;
    done : BOOL;
    ProbeDoneWhen : INT;
END_VAR
VAR_INST
    _noOfAttmets : INT;
    _timer : ton;
END_VAR
seq REF= _sequenceTixonVibro;
seq.Open();
seq.Observer := _observerTixonVibro;
_tixonPickVibroFeeder.CyclicBufferFeed();
_tixonPickVibroFeeder.CyclicBinFeed();
_tixonPickVibroFeeder.CyclicHopperFeed();
_tixonPickVibroFeeder.DefaultSignalisation();
_actualAttempt := _noOfAttmets;

IF (seq.Step(inStepID := 0, inEnabled := TRUE, inStepDescription := 'READY TO START')) THEN
    //--------------------------------------------------------
    _noOfAttmets := 0;

    answer := _dialogTixon.Show()
        .WithType(eDialogType.Question)
        .WithCaption('Ready to go?')
        .WithText('Do you really want to start feeding? Do we go ahead?')
        .WithYesNo().Answer;

    //
    IF (answer = TcoCore.eDialogAnswer.Yes) THEN
        seq.CompleteStep();
    ELSIF (answer = TcoCore.eDialogAnswer.No) THEN
        _sequenceTixonPickVibroTask.Restore();
    END_IF;
    //--------------------------------------------------------
END_IF;

IF (seq.Step(inStepID := 10, inEnabled := TRUE, inStepDescription := 'RESTORE')) THEN
    //--------------------------------------------------------
    _tixonPickVibroFeeder.Restore();
    seq.CompleteStep();
    //--------------------------------------------------------
END_IF;

IF (seq.Step(inStepID := 11, inEnabled := TRUE, inStepDescription := 'START FEEDING TASK')) THEN
    //--------------------------------------------------------
    seq.StepCompleteWhen(_tixonPickVibroFeeder.Separe().Done);
    //--------------------------------------------------------
END_IF;

IF (seq.Step(inStepID := 12, inEnabled := TRUE, inStepDescription := 'WAIT FOR COMPONENT')) THEN
    //--------------------------------------------------------
    IF _tixonPickVibroFeeder.Status.ComponentReady THEN
        seq.CompleteStep();
        _timer(IN := FALSE);
    END_IF;
    //--------------------------------------------------------
END_IF;

IF (seq.Step(inStepID := 13, inEnabled := TRUE, inStepDescription := 'WAIT FOR PICK - INTERUPT PICK ZONE')) THEN
    //--------------------------------------------------------
    IF _tixonPickVibroFeeder.Status.InPickZone THEN
        seq.CompleteStep();
    END_IF

    //--------------------------------------------------------
END_IF;

IF (seq.Step(inStepID := 14, inEnabled := TRUE, inStepDescription := 'WAIT FOR PICK - RELEASE PICK')) THEN
    //--------------------------------------------------------
    IF NOT _tixonPickVibroFeeder.Status.InPickZone AND NOT _tixonPickVibroFeeder.Status.SeparatorPresent THEN
        seq.CompleteStep();
    END_IF

    //--------------------------------------------------------
END_IF;

IF (seq.Step(inStepID := 16, inEnabled := TRUE, inStepDescription := 'COUNT')) THEN
    //--------------------------------------------------------
    IF _noOfAttmets < _maxAllowedAttemptsTixonPickVibro THEN
        _noOfAttmets := _noOfAttmets + 1;
        seq.RequestStep(11);
    ELSE
        seq.CompleteStep();
    end_if;
    //--------------------------------------------------------
END_IF;

IF (seq.Step(inStepID := 600, inEnabled := TRUE, inStepDescription := 'ASKING FOR RESTORING')) THEN
    //    --------------------------------------------------------
    _tixonPickVibroFeeder.Restore();
    answer := _dialogTixon.Show().WithType(eDialogType.Question).WithCaption('Question?').WithText('Do you want to repat it?').WithYesNo().Answer;

    IF (answer = TcoCore.eDialogAnswer.Yes) THEN
        seq.CompleteStep();
    ELSIF (answer = TcoCore.eDialogAnswer.No) THEN
        _sequenceTixonPickVibroTask.Restore();
    END_IF;
    //    --------------------------------------------------------
END_IF;

IF (seq.Step(inStepID := seq.RESTORE_STEP_ID, inEnabled := TRUE, inStepDescription := 'RETURN TO THE START OF THE SEQUENCE')) THEN
    //--------------------------------------------------------
    seq.CompleteSequence();
    //--------------------------------------------------------
END_IF;

seq.Close();
END_METHOD

METHOD SequenceTixonPickVibroBasic
VAR
    seq : REFERENCE TO TcoCore.TcoSequence;
    answer : TcoCore.eDialogAnswer;
    done : BOOL;
    ProbeDoneWhen : INT;
END_VAR
VAR_INST
    _noOfAttmets : INT;
    _timer : ton;
END_VAR
seq REF= _sequenceTixonPickVibroBasic;
seq.Open();
seq.Observer := _observerTixonPickVibroBasic;
_tixonPickVibroBasicFeeder.CyclicBufferFeed();
_tixonPickVibroBasicFeeder.CyclicHopperFeed();
_tixonPickVibroBasicFeeder.DefaultSignalisation();
_actualAttempt := _noOfAttmets;

IF (seq.Step(inStepID := 0, inEnabled := TRUE, inStepDescription := 'READY TO START')) THEN
    //--------------------------------------------------------
    _noOfAttmets := 0;

    answer := _dialogTixon.Show()
        .WithType(eDialogType.Question)
        .WithCaption('Ready to go?')
        .WithText('Do you really want to start feeding? Do we go ahead?')
        .WithYesNo().Answer;

    //
    IF (answer = TcoCore.eDialogAnswer.Yes) THEN
        seq.CompleteStep();
    ELSIF (answer = TcoCore.eDialogAnswer.No) THEN
        _tixonPickVibroBasicFeeder.Restore();
    END_IF;
    //--------------------------------------------------------
END_IF;

IF (seq.Step(inStepID := 10, inEnabled := TRUE, inStepDescription := 'RESTORE')) THEN
    //--------------------------------------------------------
    _tixonPickVibroBasicFeeder.Restore();
    seq.CompleteStep();
    //--------------------------------------------------------
END_IF;

IF (seq.Step(inStepID := 11, inEnabled := TRUE, inStepDescription := 'START FEEDING TASK')) THEN
    //--------------------------------------------------------
    seq.StepCompleteWhen(_tixonPickVibroBasicFeeder.Separe().Done);
    //--------------------------------------------------------
END_IF;

IF (seq.Step(inStepID := 12, inEnabled := TRUE, inStepDescription := 'WAIT FOR COMPONENT')) THEN
    //--------------------------------------------------------
    IF _tixonPickVibroBasicFeeder.Status.ComponentReady THEN
        seq.CompleteStep();
        _timer(IN := FALSE);
    END_IF;
    //--------------------------------------------------------
END_IF;

IF (seq.Step(inStepID := 13, inEnabled := TRUE, inStepDescription := 'WAIT FOR PICK - INTERUPT PICK ZONE')) THEN
    //--------------------------------------------------------
    IF _tixonPickVibroBasicFeeder.Status.InPickZone THEN
        seq.CompleteStep();
    END_IF

    //--------------------------------------------------------
END_IF;

IF (seq.Step(inStepID := 14, inEnabled := TRUE, inStepDescription := 'WAIT FOR PICK - RELEASE PICK')) THEN
    //--------------------------------------------------------
    IF NOT _tixonPickVibroBasicFeeder.Status.InPickZone AND NOT _tixonPickVibroBasicFeeder.Status.SeparatorPresent THEN
        seq.CompleteStep();
    END_IF

    //--------------------------------------------------------
END_IF;

IF (seq.Step(inStepID := 16, inEnabled := TRUE, inStepDescription := 'COUNT')) THEN
    //--------------------------------------------------------
    IF _noOfAttmets < _maxAllowedAttemptsTixonPickVibroBasic THEN
        _noOfAttmets := _noOfAttmets + 1;
        seq.RequestStep(11);
    ELSE
        seq.CompleteStep();
    end_if;
    //--------------------------------------------------------
END_IF;

IF (seq.Step(inStepID := 600, inEnabled := TRUE, inStepDescription := 'ASKING FOR RESTORING')) THEN
    //    --------------------------------------------------------
    _tixonPickVibroBasicFeeder.Restore();
    answer := _dialogTixon.Show().WithType(eDialogType.Question).WithCaption('Question?').WithText('Do you want to repat it?').WithYesNo().Answer;

    IF (answer = TcoCore.eDialogAnswer.Yes) THEN
        seq.CompleteStep();
    ELSIF (answer = TcoCore.eDialogAnswer.No) THEN
        _tixonPickVibroBasicFeeder.Restore();
    END_IF;
    //    --------------------------------------------------------
END_IF;

IF (seq.Step(inStepID := seq.RESTORE_STEP_ID, inEnabled := TRUE, inStepDescription := 'RETURN TO THE START OF THE SEQUENCE')) THEN
    //--------------------------------------------------------
    seq.CompleteSequence();
    //--------------------------------------------------------
END_IF;

seq.Close();
END_METHOD

METHOD SequenceTixonStep
VAR
    seq : REFERENCE TO TcoCore.TcoSequence;
    answer : TcoCore.eDialogAnswer;
    done : BOOL;
    ProbeDoneWhen : INT;
END_VAR
VAR_INST
    _noOfAttmets : INT;
    _timer : ton;
END_VAR
seq REF= _sequenceTixonStep;
seq.Open();
seq.Observer := _observerTixonStep;
_tixonStepFeeder.CyclicBufferFeed();
_tixonStepFeeder.CyclicStepperFeed();
_tixonStepFeeder.CyclicHopperFeed();
_tixonStepFeeder.DefaultSignalisation();
_actualAttempt := _noOfAttmets;

IF (seq.Step(inStepID := 0, inEnabled := TRUE, inStepDescription := 'READY TO START')) THEN
    //--------------------------------------------------------
    _noOfAttmets := 0;

    answer := _dialogTixon.Show()
        .WithType(eDialogType.Question)
        .WithCaption('Ready to go?')
        .WithText('Do you really want to start feeding? Do we go ahead?')
        .WithYesNo().Answer;

    //
    IF (answer = TcoCore.eDialogAnswer.Yes) THEN
        seq.CompleteStep();
    ELSIF (answer = TcoCore.eDialogAnswer.No) THEN
        _sequenceTixonStepTask.Restore();
    END_IF;
    //--------------------------------------------------------
END_IF;

IF (seq.Step(inStepID := 10, inEnabled := TRUE, inStepDescription := 'RESTORE')) THEN
    //--------------------------------------------------------
    _tixonStepFeeder.Restore();
    seq.CompleteStep();
    //--------------------------------------------------------
END_IF;

IF (seq.Step(inStepID := 11, inEnabled := TRUE, inStepDescription := 'START FEEDING TASK')) THEN
    //--------------------------------------------------------
    seq.StepCompleteWhen(_tixonStepFeeder.Separe().Done);
    _timer(IN := FALSE);
    //--------------------------------------------------------
END_IF;

IF (seq.Step(inStepID := 12, inEnabled := TRUE, inStepDescription := 'WAIT FOR COMPONENT AND WAITING FOR SIMULATED PROCESS')) THEN
    //--------------------------------------------------------
    _timer(IN := TRUE, PT := _estimatedCycleTime);

    IF _tixonStepFeeder.Status.ComponentReady AND _timer.Q THEN
        seq.CompleteStep();
        _timer(IN := FALSE);
    END_IF;
    //--------------------------------------------------------
END_IF;

IF (seq.Step(inStepID := 13, inEnabled := TRUE, inStepDescription := 'NASTREL')) THEN
    //--------------------------------------------------------
    _timer(IN := TRUE, PT := _pushTime);
    _tixonStepFeeder.Push(TRUE);

    IF _timer.Q THEN
        seq.CompleteStep();
        _tixonStepFeeder.Push(FALSE);
    END_IF;
    //--------------------------------------------------------
END_IF;

IF (seq.Step(inStepID := 16, inEnabled := TRUE, inStepDescription := 'COUNT')) THEN
    //--------------------------------------------------------
    IF _noOfAttmets < _maxAllowedAttemptsTixonStep THEN
        _noOfAttmets := _noOfAttmets + 1;
        seq.RequestStep(11);
    ELSE
        seq.CompleteStep();
    end_if;
    //--------------------------------------------------------
END_IF;

IF (seq.Step(inStepID := 600, inEnabled := TRUE, inStepDescription := 'ASKING FOR RESTORING')) THEN
    //    --------------------------------------------------------
    _tixonStepFeeder.Restore();
    answer := _dialogTixon.Show().WithType(eDialogType.Question).WithCaption('Question?').WithText('Do you want to repat it?').WithYesNo().Answer;

    IF (answer = TcoCore.eDialogAnswer.Yes) THEN
        seq.CompleteStep();
    ELSIF (answer = TcoCore.eDialogAnswer.No) THEN
        _sequenceTixonStepTask.Restore();
    END_IF;
    //    --------------------------------------------------------
END_IF;

IF (seq.Step(inStepID := seq.RESTORE_STEP_ID, inEnabled := TRUE, inStepDescription := 'RETURN TO THE START OF THE SEQUENCE')) THEN
    //--------------------------------------------------------
    seq.CompleteSequence();
    //--------------------------------------------------------
END_IF;

seq.Close();
END_METHOD

METHOD SequenceTixonVibro
VAR
    seq : REFERENCE TO TcoCore.TcoSequence;
    answer : TcoCore.eDialogAnswer;
    done : BOOL;
    ProbeDoneWhen : INT;
END_VAR
VAR_INST
    _noOfAttmets : INT;
    _timer : ton;
END_VAR
seq REF= _sequenceTixonVibro;
seq.Open();
seq.Observer := _observerTixonVibro;
_tixonVibroFeeder.CyclicBufferFeed();
_tixonVibroFeeder.CyclicHopperFeed();
_tixonVibroFeeder.DefaultSignalisation();
_actualAttempt := _noOfAttmets;

IF (seq.Step(inStepID := 0, inEnabled := TRUE, inStepDescription := 'READY TO START')) THEN
    //--------------------------------------------------------
    _noOfAttmets := 0;

    answer := _dialogTixon.Show()
        .WithType(eDialogType.Question)
        .WithCaption('Ready to go?')
        .WithText('Do you really want to start feeding? Do we go ahead?')
        .WithYesNo().Answer;

    //
    IF (answer = TcoCore.eDialogAnswer.Yes) THEN
        seq.CompleteStep();
    ELSIF (answer = TcoCore.eDialogAnswer.No) THEN
        _sequenceTixonVibroTask.Restore();
    END_IF;
    //--------------------------------------------------------
END_IF;

IF (seq.Step(inStepID := 10, inEnabled := TRUE, inStepDescription := 'RESTORE')) THEN
    //--------------------------------------------------------
    _tixonVibroFeeder.Restore();
    seq.CompleteStep();
    //--------------------------------------------------------
END_IF;

IF (seq.Step(inStepID := 11, inEnabled := TRUE, inStepDescription := 'START FEEDING TASK')) THEN
    //--------------------------------------------------------
    seq.StepCompleteWhen(_tixonVibroFeeder.Separe().Done);
    _timer(IN := FALSE);
    //--------------------------------------------------------
END_IF;

IF (seq.Step(inStepID := 12, inEnabled := TRUE, inStepDescription := 'WAIT FOR COMPONENT AND WAITING FOR SIMULATED PROCESS')) THEN
    //--------------------------------------------------------
    _timer(IN := TRUE, PT := _estimatedCycleTime);

    IF _tixonVibroFeeder.Status.ComponentReady AND _timer.Q THEN
        seq.CompleteStep();
        _timer(IN := FALSE);
    END_IF;
    //--------------------------------------------------------
END_IF;

IF (seq.Step(inStepID := 13, inEnabled := TRUE, inStepDescription := 'NASTREL')) THEN
    //--------------------------------------------------------
    _timer(IN := TRUE, PT := _pushTime);
    _tixonVibroFeeder.Push(TRUE);

    IF _timer.Q THEN
        seq.CompleteStep();
        _tixonVibroFeeder.Push(FALSE);
    END_IF;
    //--------------------------------------------------------
END_IF;

IF (seq.Step(inStepID := 16, inEnabled := TRUE, inStepDescription := 'COUNT')) THEN
    //--------------------------------------------------------
    IF _noOfAttmets < _maxAllowedAttemptsTixonVibro THEN
        _noOfAttmets := _noOfAttmets + 1;
        seq.RequestStep(11);
    ELSE
        seq.CompleteStep();
    end_if;
    //--------------------------------------------------------
END_IF;

IF (seq.Step(inStepID := 600, inEnabled := TRUE, inStepDescription := 'ASKING FOR RESTORING')) THEN
    //    --------------------------------------------------------
    _tixonVibroFeeder.Restore();
    answer := _dialogTixon.Show().WithType(eDialogType.Question).WithCaption('Question?').WithText('Do you want to repat it?').WithYesNo().Answer;

    IF (answer = TcoCore.eDialogAnswer.Yes) THEN
        seq.CompleteStep();
    ELSIF (answer = TcoCore.eDialogAnswer.No) THEN
        _sequenceTixonVibroTask.Restore();
    END_IF;
    //    --------------------------------------------------------
END_IF;

IF (seq.Step(inStepID := seq.RESTORE_STEP_ID, inEnabled := TRUE, inStepDescription := 'RETURN TO THE START OF THE SEQUENCE')) THEN
    //--------------------------------------------------------
    seq.CompleteSequence();
    //--------------------------------------------------------
END_IF;

seq.Close();
END_METHOD

END_FUNCTION_BLOCK

// ---- Tests/TcoContext/SequenceTask.TcPOU
FUNCTION_BLOCK SequenceTask EXTENDS TcoCore.TcoTask
VAR_INPUT
    Sequence : TcoCore.ITcoSequencer;
END_VAR

(*~
    <docu>
        <summary>
            Restores this instance to the Ready state. Can be called explicitly or from within one of the restore mechanisms.
            <para>
                See also <see cref="PlcDocu.TcoCore.TcoTask.AutoRestorable()"/>
            </para>
        </summary>
    </docu>
~*)
METHOD Restore : ITcoRestorable
SUPER^.Restore();
THIS^.Sequence.Restore();
END_METHOD

END_FUNCTION_BLOCK
